// TIA Portal V20 export
TYPE "LER_typeQrReadTrackingData"
// stored: Access Published
   STRUCT
      resultData { ExternalWritable := 'False'} : String[31];
      resultOK { ExternalWritable := 'False'} : Bool;
      resultNG { ExternalWritable := 'False'} : Bool;
      complete { ExternalWritable := 'False'} : Bool;
   END_STRUCT;
END_TYPE
